{attribute 'GeneratedUsingTerminal: EL2911-0000-0016'}
{attribute addProperty BoxType "EL2911-0000-0016"}
{attribute addProperty Id "FIELDVOLTAGE_Field_Voltage_StatusFIELDVOLTAGE_Field_Voltage_Status_9DC7C3492"}
{attribute addProperty CRC "1604760807"}
{attribute addProperty Size "2"}
TYPE Module_3_DEVICEIO_5FA6B4E7 :
STRUCT
	{attribute addProperty Name "FIELDVOLTAGE_Field_Voltage_Status"}
	FIELDVOLTAGE_Field_Voltage_Status  : FIELDVOLTAGE_Field_Voltage_Status_9DC7C349;
END_STRUCT
END_TYPE

(* stored: Version 1.2.0.0, ProductVersion 3.1.4024.9
   DUT Module_3_DEVICEIO_5FA6B4E7: Id {1e9f0b60-078d-4ef0-ab71-fd00361f1bf6} *)
